// TIA Portal V16 export
// export: Created 2024-05-11T02:56:22.7501852Z, ExportSetting WithDefaults, DisplayName Totally Integrated Automation Portal, DisplayVersion V16, DisplayName TIA Portal Version Control Interface, DisplayVersion V16, DisplayName TIA Portal Openness, DisplayVersion V16, DisplayName STEP 7 Professional, DisplayVersion V16, DisplayName STEP 7 Safety, DisplayVersion V16, DisplayName WinCC Professional, DisplayVersion V16
FUNCTION_BLOCK "K21_ST09上自动"   // FB21, LAD
{ S7_Optimized_Access := 'TRUE' }
VERSION : 0.1
// stored: AutoNumber false, IsIECCheckEnabled false, IsRetainMemResEnabled false, MemoryReserve 100, SetENOAutomatically false, UDAEnableTagReadback false
   VAR_TEMP   // added for the SCL form of the ladder/FBD networks
      _w1 : Bool;
   END_VAR
BEGIN

REGION Network 2: @搬出条件，SN11===ST09上工位
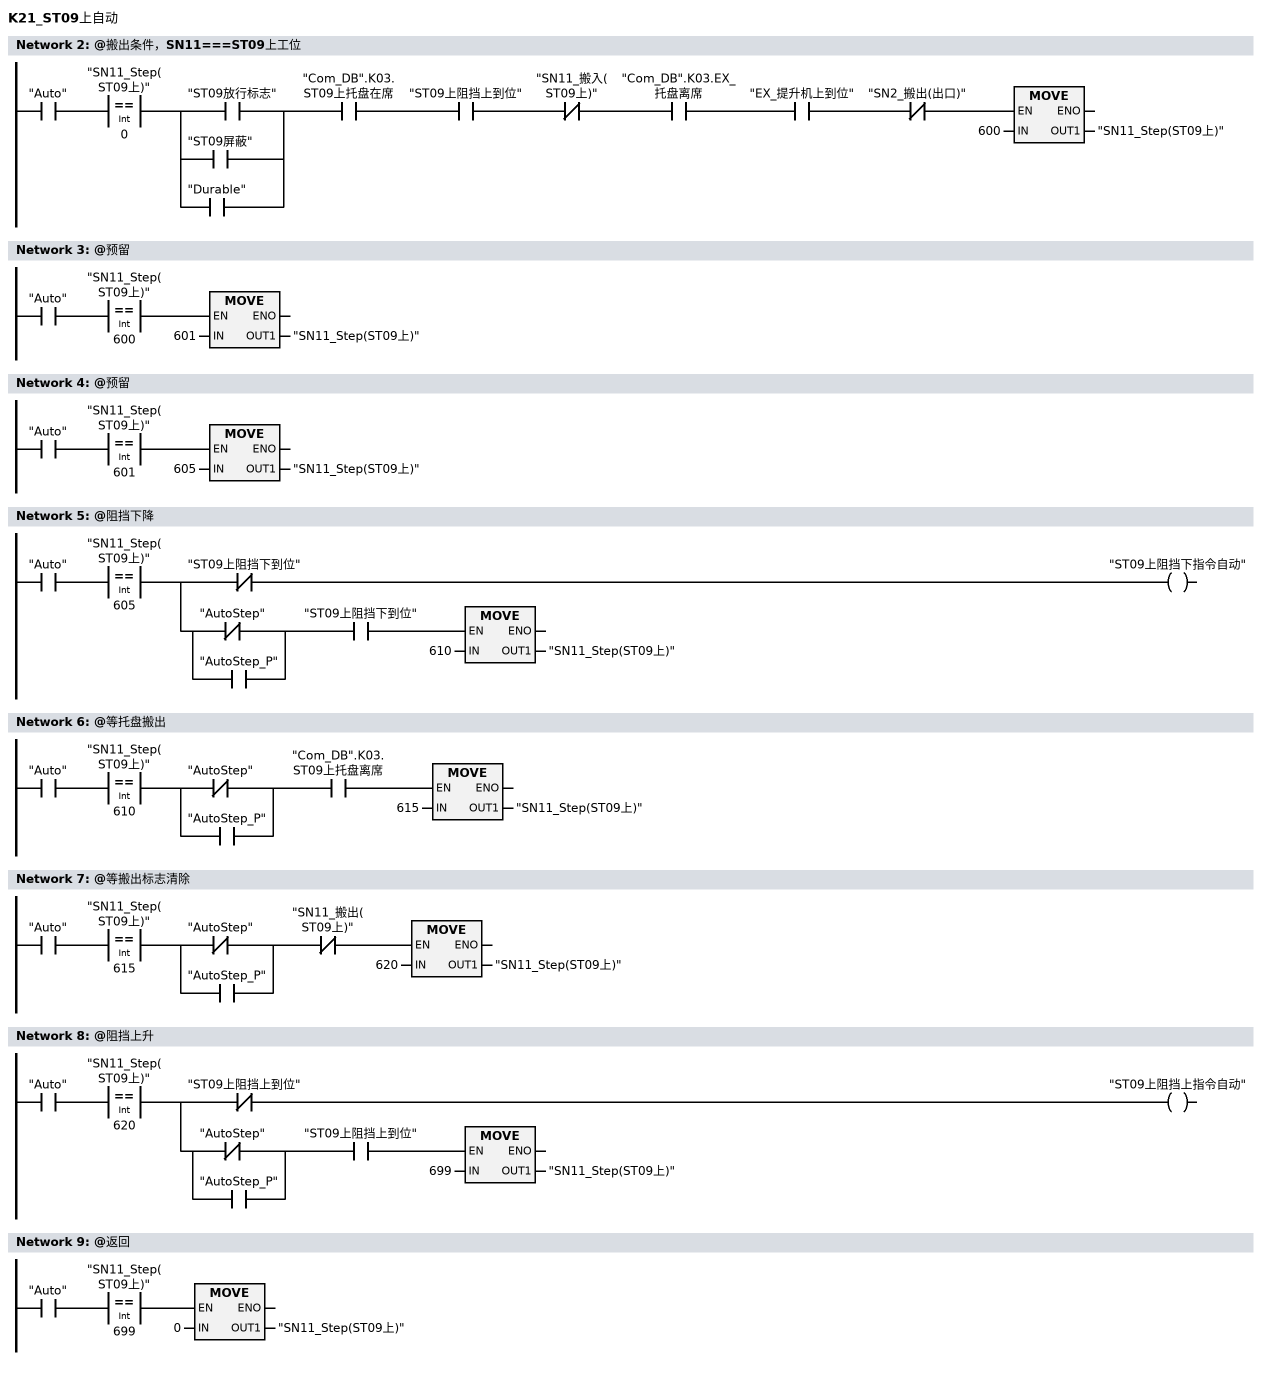
   RUNG wire#powerrail
      Contact( "Auto" )
      { S7_Templates := "SrcType := Int" } EQ_Contact(in1 := "SN11_Step(ST09上)", in2 := 0)
      wire#w1
      Contact( "ST09放行标志" )
      wire#w2
      Contact( "Com_DB".K03.ST09上托盘在席 )
      Contact( "ST09上阻挡上到位" )
      I_Contact( "SN11_搬入(ST09上)" )
      Contact( "Com_DB".K03.EX_托盘离席 )
      Contact( "EX_提升机上到位" )
      I_Contact( "SN2_搬出(出口)" )
      Move(in := 600, out1 => "SN11_Step(ST09上)")
   END_RUNG
   RUNG wire#w1
      Contact( "ST09屏蔽" )
   END_RUNG wire#w2
   RUNG wire#w1
      Contact( "Durable" )
   END_RUNG wire#w2
   // the same network as SCL:
   IF "Auto" AND ("SN11_Step(ST09上)" = 0) AND ("ST09放行标志" OR "ST09屏蔽" OR "Durable") AND "Com_DB".K03.ST09上托盘在席 AND "ST09上阻挡上到位" AND NOT "SN11_搬入(ST09上)" AND "Com_DB".K03.EX_托盘离席 AND "EX_提升机上到位" AND NOT "SN2_搬出(出口)" THEN
       "SN11_Step(ST09上)" := 600;
   END_IF;
END_REGION

REGION Network 3: @预留
   RUNG wire#powerrail
      Contact( "Auto" )
      { S7_Templates := "SrcType := Int" } EQ_Contact(in1 := "SN11_Step(ST09上)", in2 := 600)
      Move(in := 601, out1 => "SN11_Step(ST09上)")
   END_RUNG
   // the same network as SCL:
   IF "Auto" AND ("SN11_Step(ST09上)" = 600) THEN "SN11_Step(ST09上)" := 601; END_IF;
END_REGION

REGION Network 4: @预留
   RUNG wire#powerrail
      Contact( "Auto" )
      { S7_Templates := "SrcType := Int" } EQ_Contact(in1 := "SN11_Step(ST09上)", in2 := 601)
      Move(in := 605, out1 => "SN11_Step(ST09上)")
   END_RUNG
   // the same network as SCL:
   IF "Auto" AND ("SN11_Step(ST09上)" = 601) THEN "SN11_Step(ST09上)" := 605; END_IF;
END_REGION

REGION Network 5: @阻挡下降
   RUNG wire#powerrail
      Contact( "Auto" )
      { S7_Templates := "SrcType := Int" } EQ_Contact(in1 := "SN11_Step(ST09上)", in2 := 605)
      wire#w1
      I_Contact( "ST09上阻挡下到位" )
      Coil( "ST09上阻挡下指令自动" )
   END_RUNG
   RUNG wire#w1
      I_Contact( "AutoStep" )
      wire#w2
      Contact( "ST09上阻挡下到位" )
      Move(in := 610, out1 => "SN11_Step(ST09上)")
   END_RUNG
   RUNG wire#w1
      Contact( "AutoStep_P" )
   END_RUNG wire#w2
   // the same network as SCL:
   #_w1 := "Auto" AND ("SN11_Step(ST09上)" = 605);
   "ST09上阻挡下指令自动" := #_w1 AND NOT "ST09上阻挡下到位";
   IF #_w1 AND (NOT "AutoStep" OR "AutoStep_P") AND "ST09上阻挡下到位" THEN "SN11_Step(ST09上)" := 610; END_IF;
END_REGION

REGION Network 6: @等托盘搬出
   RUNG wire#powerrail
      Contact( "Auto" )
      { S7_Templates := "SrcType := Int" } EQ_Contact(in1 := "SN11_Step(ST09上)", in2 := 610)
      wire#w1
      I_Contact( "AutoStep" )
      wire#w2
      Contact( "Com_DB".K03.ST09上托盘离席 )
      Move(in := 615, out1 => "SN11_Step(ST09上)")
   END_RUNG
   RUNG wire#w1
      Contact( "AutoStep_P" )
   END_RUNG wire#w2
   // the same network as SCL:
   IF "Auto" AND ("SN11_Step(ST09上)" = 610) AND (NOT "AutoStep" OR "AutoStep_P") AND "Com_DB".K03.ST09上托盘离席 THEN
       "SN11_Step(ST09上)" := 615;
   END_IF;
END_REGION

REGION Network 7: @等搬出标志清除
   RUNG wire#powerrail
      Contact( "Auto" )
      { S7_Templates := "SrcType := Int" } EQ_Contact(in1 := "SN11_Step(ST09上)", in2 := 615)
      wire#w1
      I_Contact( "AutoStep" )
      wire#w2
      I_Contact( "SN11_搬出(ST09上)" )
      Move(in := 620, out1 => "SN11_Step(ST09上)")
   END_RUNG
   RUNG wire#w1
      Contact( "AutoStep_P" )
   END_RUNG wire#w2
   // the same network as SCL:
   IF "Auto" AND ("SN11_Step(ST09上)" = 615) AND (NOT "AutoStep" OR "AutoStep_P") AND NOT "SN11_搬出(ST09上)" THEN
       "SN11_Step(ST09上)" := 620;
   END_IF;
END_REGION

REGION Network 8: @阻挡上升
   RUNG wire#powerrail
      Contact( "Auto" )
      { S7_Templates := "SrcType := Int" } EQ_Contact(in1 := "SN11_Step(ST09上)", in2 := 620)
      wire#w1
      I_Contact( "ST09上阻挡上到位" )
      Coil( "ST09上阻挡上指令自动" )
   END_RUNG
   RUNG wire#w1
      I_Contact( "AutoStep" )
      wire#w2
      Contact( "ST09上阻挡上到位" )
      Move(in := 699, out1 => "SN11_Step(ST09上)")
   END_RUNG
   RUNG wire#w1
      Contact( "AutoStep_P" )
   END_RUNG wire#w2
   // the same network as SCL:
   #_w1 := "Auto" AND ("SN11_Step(ST09上)" = 620);
   "ST09上阻挡上指令自动" := #_w1 AND NOT "ST09上阻挡上到位";
   IF #_w1 AND (NOT "AutoStep" OR "AutoStep_P") AND "ST09上阻挡上到位" THEN "SN11_Step(ST09上)" := 699; END_IF;
END_REGION

REGION Network 9: @返回
   RUNG wire#powerrail
      Contact( "Auto" )
      { S7_Templates := "SrcType := Int" } EQ_Contact(in1 := "SN11_Step(ST09上)", in2 := 699)
      Move(in := 0, out1 => "SN11_Step(ST09上)")
   END_RUNG
   // the same network as SCL:
   IF "Auto" AND ("SN11_Step(ST09上)" = 699) THEN "SN11_Step(ST09上)" := 0; END_IF;
END_REGION
END_FUNCTION_BLOCK
